(* Logix 5000 project; controller studio_5000_first_program Emulate 5570 rev 30.12; software revision 30.01 *)

TASK MainTask (continuous, watchdog 500 ms) : MainProgram

MODULES
   Local : Emulate 5570 (ICP 2, rev 30.12)
END_MODULES

PROGRAM MainProgram   (* main routine MainRoutine *)
VAR
   Motor : BOOL;
   Star : BOOL;
   Stop : BOOL;
END_VAR

ROUTINE MainRoutine   (* ladder *)
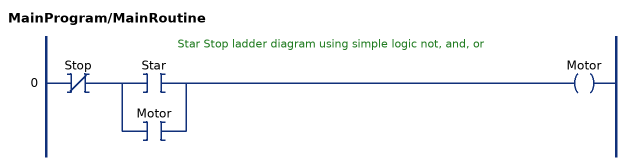
   // Star Stop ladder diagram using simple logic not, and, or
   0: XIO(Stop)[XIC(Star) ,XIC(Motor) ]OTE(Motor);
END_ROUTINE
END_PROGRAM
